Universal Robots PolyScope program: create_cotton_candy123trashy.urp

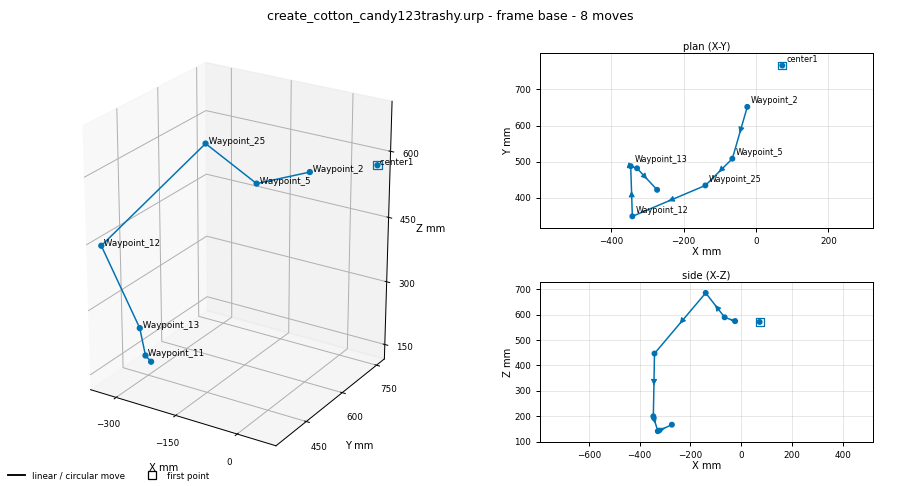
[picture p0: tool path of create_cotton_candy123trashy.urp in frame base, 8 of 14 moves have a stored position in this frame; points joined in program order, loops and branches not executed]
Program create_cotton_candy123trashy (installation=default directory=/programs/Nicolas_Arteaga/Old createdIn=5.8.2.10297 lastSavedIn=5.12.4.1101661 robotSerialNumber=20225502378)
Calibrated DH parameters: a=[0.00022, -0.425328, -0.389701, 0.000059, 0.000065, 0]; d=[0.162608, 0.803456, 9.992211, -10.662202, 0.099702, 0.099559]; alpha=[1.570756, 0.001543, 0.004316, 1.570651, -1.570122, 0]; deltaTheta=[0, 0.002917, 0.116094, -0.119008, 0, -0.000001]
Robot Program (runOnlyOnce=true)
  MoveL speed 250 mm/s, acceleration 1200 mm/s^2 (useActiveTCP=true) feature=Base
    Waypoint center1: TCP in base x=72.723 y=766.045 z=571.175 mm, rx=-1.5688 ry=-0.0203 rz=0.0146 rad; joints [244.553, -79.065, 65.7, 13.074, 63.165, 180.144] deg; TCP offset x=0 y=0 z=191.5 mm, rx=0 ry=0 rz=0 rad
  'Now Cotton Candy Creation'
  SuppressedNode
    radius := 0.149
  radius := 0.14
  height := 0.05
  SuppressedNode
    cold_start_wait := 101.25
  SuppressedNode
    start_wait := GP_int_in[0]
  SuppressedNode
    start_time := GP_int_in[1]
  SuppressedNode
    circle_time := GP_int_in[2]
  start_wait := 1
  start_time := 33.75
  circle_time := 3.75
  SuppressedNode
    cold_start_spin := 28
  SuppressedNode
    cold_start_spin := 100
  center := Joint_6_name
  bottom := pose_add(center, p[0, -radius, height, 0, 0, 0])
  right := pose_add(center, p[-radius, 0, -height, 0, 0, 0])
  top_circ := pose_add(center, p[0, radius, height, 0, 0, 0])
  left := pose_add(center, p[radius, 0, -height, 0, 0, 0])
  SuppressedNode
    Wait Sleep waitTime=101.25
  SuppressedNode
    Wait Condition expression=GP_int_in[0]
  Script: sleep(start_wait)
  Loop While (checkContinuously=false) expression=start_time>0
    MoveP speed 250 mm/s, acceleration 1200 mm/s^2 (blendRadius=0.125 useActiveTCP=true) feature=Base
      Waypoint Waypoint (Variable): variable(name=bottom)
      CircleMove (OrientationMode=UNCONSTRAINED)
        Waypoint Waypoint (Variable): variable(name=left)
        Waypoint Waypoint (Variable): variable(name=top_circ)
    MoveP speed 250 mm/s, acceleration 1200 mm/s^2 (blendRadius=0.025 useActiveTCP=true) feature=Base
      Waypoint Waypoint (Variable): variable=top_circ
      CircleMove (OrientationMode=UNCONSTRAINED)
        Waypoint Waypoint (Variable): variable(name=right)
        Waypoint Waypoint (Variable): variable=bottom
  MoveL speed 250 mm/s, acceleration 1200 mm/s^2 (useActiveTCP=true) feature=Base
    Waypoint Waypoint_2: TCP in base x=-24.03 y=651.793 z=574.352 mm, rx=-0.9882 ry=-1.0644 rz=-1.2372 rad; joints [248.909, -99.854, 96.502, -11.42, 64.977, 96.89] deg
    Waypoint Waypoint_5: TCP in base x=-65.345 y=508.583 z=589.478 mm, rx=-0.8529 ry=-1.3704 rz=-1.3892 rad; joints [239.18, -119.542, 101.662, 8.745, 51.039, 78.082] deg
    Waypoint Waypoint_25: TCP in base x=-139.92 y=434.562 z=685.517 mm, rx=0.2728 ry=-1.6358 rz=-2.1043 rad; joints [228.521, -129.991, 99.843, -7.046, 27.223, 41.249] deg
    Waypoint Waypoint_12: TCP in base x=-341.731 y=349.139 z=446.744 mm, rx=1.0197 ry=-1.4327 rz=-1.9509 rad; joints [261.046, -128.059, 128.66, -21.395, 27.658, 2.719] deg
    Waypoint Waypoint_13: TCP in base x=-346.288 y=487.83 z=199.367 mm, rx=1.1258 ry=-1.8238 rz=-1.9724 rad; joints [274.508, -89.471, 132.703, -38.479, 53.378, -24.773] deg
    Waypoint Waypoint_11: TCP in base x=-328.73 y=482.036 z=140.622 mm, rx=1.1107 ry=-1.8448 rz=-1.9801 rad; joints [271.637, -83.004, 138.617, -50.548, 51.741, -25.068] deg
    URCap Gripper Activate (Robotiq_Grippers, Robotiq Inc.) dataModel(ResetAndActivateKey=false)
    URCap Gripper (Robotiq_Grippers, Robotiq Inc.) dataModel(position=0.0, force=0.0, speed=100.0, positionInDouble=0.0, forceInDouble=0.0, speedInDouble=100.0, slaveIds=[9], blocking=true)
    Waypoint Waypoint_14: TCP in base x=-273.276 y=422.463 z=166.295 mm, rx=0.9524 ry=-2.167 rz=-1.9141 rad; joints [271.624, -104.005, 143.852, -26.72, 64.174, -25.036] deg
    URCap Gripper (Robotiq_Grippers, Robotiq Inc.) dataModel(position=100.0, force=0.0, speed=100.0, positionInDouble=100.0, forceInDouble=0.0, speedInDouble=100.0, slaveIds=[9], blocking=true)
